Staubli VAL3: Axis8OnReady.pgx

public program Axis8OnReady(num x_nPosition (dimensions=1), num x_nSpeed (dimensions=1), num x_nPrecent (dimensions=1), bool& x_bRes (dimensions=1))
  local bool l_bBool
  local num l_nNum
begin


  //异步八轴到位
  x_bRes=false

  //参数合法性
  if x_nSpeed<=0 or x_nPrecent<=0 or x_nPosition<=0
    return
  endIf



  //没有电或者报警
  if dDio["In4_b8MotorPower"]==false or dDio["In4_b8MotorError"]==true or dDio["In4_b8BackHome"]==false
    return
  endIf

  call AxisIsNeg(true,l_bBool)
  if l_bBool
    return
  endIf


  dDio["O4_b8RecordPos"]=true
  delay(0.2)
  dDio["O4_b8RecordPos"]=false

  call GetAxis8Pos(l_nNum,x_nPrecent)

  if abs(l_nNum-x_nPosition)!=0
    waitEndMove()
  else
    x_bRes=true
    return
  endIf

  dDio["O4_b8StopMotor"]=false
  delay(0.2)
  x_nPosition=x_nPosition*x_nPrecent
  aioSet(aAio["O4_a8Velocity"],max(1,x_nSpeed*x_nPrecent*16.666667))
  aioSet(aAio["O4_a8MovePosL"],x_nPosition%power(2,16))
  aioSet(aAio["O4_a8MovePosH"],roundDown(x_nPosition/power(2,16)))
  dDio["O4_b8MoveToPos"]=true
  delay(0.2)
  dDio["O4_b8MoveToPos"]=false

  x_nPosition=x_nPosition/x_nPrecent
  while dDio["In4_b8Reached"]!=true or abs(l_nNum-x_nPosition)>10
    call GetAxis8Pos(l_nNum,x_nPrecent)
    if dDio["O4_b8StopMotor"]==true
      x_bRes=false
      return
    endIf
    delay(0)
  endWhile

  x_bRes=true


end
